// TIA Portal V16 export
// export: Created 2021-07-12T14:47:21.1686958Z, ExportSetting WithDefaults, DisplayName Totally Integrated Automation Portal, DisplayVersion V16, DisplayName TIA Portal Version Control Interface, DisplayVersion V16, DisplayName TIA Portal Openness, DisplayVersion V16, DisplayName STEP 7 Professional, DisplayVersion V16, DisplayName STEP 7 Safety, DisplayVersion V16, DisplayName WinCC Professional, DisplayVersion V16
TYPE "LSimaHydTO_typeInternalControlDirectOutput"
TITLE = LSimaHydTO_typeInternalControlDirectOutput
// Manual output control
// stored: IsFailsafeCompliant false
   STRUCT
      activate : Bool;   // enables direct setting of output
      jogForward : Bool;   // direct output is active in positive direction if TRUE
      jogBackward : Bool;   // direct output is active in negative direction if TRUE
      commandValueForward : LReal := 5.0;   // direct output value in positive direction [%]
      commandValueBackward : LReal := 5.0;   // direct output value in negative direction [%]
      commandValueRamp : LReal := 100.0;   // Ramp for command value [%/s]
      offset : LReal := 0.0;   // Manipulated variable as drift compensation [%]
      safetyDistance : LReal := 50.0;   // Safety distance to avoid passing over the min. and max. positions [mm]
      commandID : UDInt;   // commanID for tracking
   END_STRUCT;
END_TYPE
